Staubli VAL3: getSetting.pgx

public program getSetting(settingType& setting_)
begin
   switch setting_.sType
        case "num"
          $exec("setting_.nValue="+setting_.varName)
        break
        case "bool"
          $exec("setting_.bValue="+setting_.varName)
        break
        case "string"
          $exec("setting_.sValue="+setting_.varName)
        break
  endSwitch
end
